TYPE FleetManagement :
STRUCT
	
	nRobotNumber			: INT;
	fSoC					: LREAL;
	nEstimatedRunningTime	: UDINT;
	ChargeRequired			: BOOL;
	
END_STRUCT
END_TYPE

(* stored: Version 1.1.0.1, ProductVersion 3.1.4024.6
   DUT FleetManagement: Id {76dff604-b5a3-4ee3-a91f-65a8a6d3681b} *)
